FUNCTION_BLOCK FB_DAU
VAR_INPUT
END_VAR
VAR_OUTPUT
END_VAR
VAR
END_VAR

METHOD PUBLIC Extend : BOOL
VAR_INPUT
END_VAR
END_METHOD

METHOD PUBLIC Init : BOOL
VAR_INPUT
END_VAR
END_METHOD

METHOD PUBLIC Retract : BOOL
VAR_INPUT
END_VAR
END_METHOD

METHOD PUBLIC TrigFault : BOOL
VAR_INPUT
END_VAR
END_METHOD

END_FUNCTION_BLOCK

(* stored: Version 1.1.0.1, ProductVersion 3.1.4022.12
   POU FB_DAU: Id {0e4ffa83-66cd-4bfb-a73f-6fc328aada0e}, SpecialFunc None
   Method Extend: Id {b84f61ca-729e-4fb1-b7e2-5667780a4e2f}
   Method Init: Id {c45dd152-7d6f-479c-963b-f1ff968fa19e}
   Method Retract: Id {b8935e9a-1ffa-4a5f-a896-3267af0042e8}
   Method TrigFault: Id {07393e28-54b7-48bc-9e2f-36ab96618aaa} *)
